// TIA Portal V19 export
TYPE "C201_STU_VLZ_TYPIC"
   STRUCT
      CMD { ExternalAccessible := 'False'; ExternalVisible := 'False'; ExternalWritable := 'False'} : USInt;   // Sturing verlichtingszone algemeen
   END_STRUCT;
END_TYPE
